{attribute 'GeneratedUsingTerminal: EK1100-0000-0018'}
{attribute addProperty BoxType "EK1100-0000-0018"}
{attribute addProperty Id "RC50_B1_EL7041_1000EL7041_86DE63E743RC50_B2_EL7041_1000EL7041_86DE63E743RC50_C11_EL7041_1000EL7041_86DE63E743RC50_C12_EL7041_1000EL7041_86DE63E743RC50_C21_EL7041_1000EL7041_86DE63E743RC50_C22_EL7041_1000EL7041_86DE63E743RC50_2_EndTerminal_EL9010EL9010_D29C20850"}
{attribute addProperty CRC "2018779948"}
{attribute addProperty Size "258"}
{attribute addProperty Name "RC50_2 (EK1100)"}
TYPE RC50_2_EK1100_7854232C EXTENDS EK1100_1FC0878B : 
STRUCT
    {attribute addProperty Name "RC50_B1 (EL7041-1000)"}
    {attribute addProperty PreviousPort "RC50_2 (EK1100) : B"}
    {attribute addProperty SyncUnit "C50"}
    RC50_B1_EL7041_1000 : EL7041_86DE63E7;
    {attribute addProperty Name "RC50_B2 (EL7041-1000)"}
    {attribute addProperty PreviousPort "RC50_B1 (EL7041-1000) : B"}
    {attribute addProperty SyncUnit "C50"}
    RC50_B2_EL7041_1000 : EL7041_86DE63E7;
    {attribute addProperty Name "RC50_C11 (EL7041-1000)"}
    {attribute addProperty PreviousPort "RC50_B2 (EL7041-1000) : B"}
    {attribute addProperty SyncUnit "C50"}
    RC50_C11_EL7041_1000 : EL7041_86DE63E7;
    {attribute addProperty Name "RC50_C12 (EL7041-1000)"}
    {attribute addProperty PreviousPort "RC50_C11 (EL7041-1000) : B"}
    {attribute addProperty SyncUnit "C50"}
    RC50_C12_EL7041_1000 : EL7041_86DE63E7;
    {attribute addProperty Name "RC50_C21 (EL7041-1000)"}
    {attribute addProperty PreviousPort "RC50_C12 (EL7041-1000) : B"}
    {attribute addProperty SyncUnit "C50"}
    RC50_C21_EL7041_1000 : EL7041_86DE63E7;
    {attribute addProperty Name "RC50_C22 (EL7041-1000)"}
    {attribute addProperty PreviousPort "RC50_C21 (EL7041-1000) : B"}
    {attribute addProperty SyncUnit "C50"}
    RC50_C22_EL7041_1000 : EL7041_86DE63E7;
    {attribute addProperty Name "RC50_2_EndTerminal (EL9010)"}
    {attribute addProperty PreviousPort "RC50_C22 (EL7041-1000) : B"}
    {attribute addProperty SyncUnit "default"}
    RC50_2_EndTerminal_EL9010 : EL9010_D29C2085;
END_STRUCT
END_TYPE

(* stored: Version 1.2.0.0, ProductVersion 3.1.4024.11
   DUT RC50_2_EK1100_7854232C: Id {db9d1586-76bd-0708-1a12-755d609a65bc} *)
